// TwinCAT 3 PLC project Untitled1
// ProgramVersion: 3.1.4023.0
// libraries:
//   Tc2_Standard, * (Beckhoff Automation GmbH)
//   Tc2_System, * (Beckhoff Automation GmbH)
//   Tc3_Module, * (Beckhoff Automation GmbH)
// project tree:
//   / PlcTask.TcTTO
//   POUs/ FB_Flasher.TcPOU, MAIN.TcPOU, PRG_1.TcPOU
// real-time tasks:
//   TASK PlcTask: cycle T#10ms, priority 20, ADS port 350

CONFIGURATION Untitled1
    RESOURCE PLC ON TwinCAT3
        TASK PlcTask(INTERVAL := T#10ms, PRIORITY := 20);
        PROGRAM MAIN WITH PlcTask : MAIN;
    END_RESOURCE
END_CONFIGURATION

// ---- POUs/MAIN.TcPOU
PROGRAM MAIN
VAR

END_VAR



PRG_1();

END_PROGRAM

// ---- POUs/PRG_1.TcPOU
PROGRAM PRG_1
VAR
	
	nState: INT;	
	
	bSignalLamp: BOOL;
	
	bSelectorSw: BOOL;
	
	bMotorStart: BOOL;
	bMotorStop: BOOL;
	
	bMotor: BOOL;

	bDelta: BOOL;
	bStar: BOOL;

	bUp: BOOL;
	bDown: BOOL;
	bRight: BOOL;
	bLeft: BOOL;

	bMotorUp: BOOL;
	bMotorDown: BOOL;
	bMotorR: BOOL;
	bMotorL: BOOL;

	bUpSW: BOOL;
	bDownLW: BOOL;
	bRightSW: BOOL;
	bLeftSW: BOOL;
	
	bLedUp: BOOL;
	bLedDown: BOOL;
	bLedR: BOOL;
	bLedL: BOOL;
	
	FlasherRight: FB_Flasher;
	FlasherLeft: FB_Flasher;
	FlasherUp: FB_Flasher;
	FlasherDown: FB_Flasher;
	FB_FlasherCurrency: FB_Flasher;
	FB_FlasherTemp: FB_Flasher;
	
	T1: TON;
	T2: TON;
	
	nValue: INT;
	bFan1: BOOL;
	bFan2: BOOL;
	bTempLamp: BOOL;
	
	
	bEmergecyStop: BOOL;
	bCurrencyLamp: BOOL;
END_VAR



ACT_1();
ACT_3();

IF T2.Q THEN
	
	ACT_2();
			
END_IF



IF bEmergecyStop THEN
	//Her şeyi sıfırla
END_IF

ACTION ACT_1:

T1(IN:=bStar , PT:=T#2M , Q=> , ET=> );
T2(IN:=bMotor , PT:=T#5M , Q=> , ET=> );

CASE nState OF

	0:
	
		IF bSelectorSw THEN
			
			bSignalLamp	:=	TRUE;
			nState := 10;
			FB_FlasherCurrency(bStart:=FALSE);
			
		END_IF
	10:
	
		IF bMotorStart AND NOT bMotorStop THEN
			
			bStar	:=	TRUE;
			bDelta	:= FALSE;
			bMotor	:=	TRUE;
			
			nState := 20;
			
		END_IF
		
	20:	
	
		IF T1.Q THEN
			
			bStar	:=	FALSE;
			bDelta	:= 	TRUE;
			
		END_IF

END_CASE

IF NOT bMotorStart AND bMotorStop	THEN
	
	nState	:=	 0;
	bMotor	:=	FALSE;
	
END_IF

IF T1.Q AND NOT bUp 
AND NOT bDown 
AND NOT bRight
AND NOT bLeft THEN 

	FB_FlasherCurrency(bStart:=TRUE , bLed=>bCurrencyLamp );
	bMotor	:=	FALSE;
	nState	:=	0;
	
END_IF
END_ACTION

ACTION ACT_2:

//LimitSW ler NC olduğu kabul edilmiştir.

FlasherUp(bStart:=bMotorUp , bLed=>bLedUp );
FlasherDown(bStart:=bMotorDown , bLed=>bLedDown );

FlasherRight(bStart:=bMotorR , bLed=>bLedR );
FlasherLeft(bStart:=bMotorL , bLed=>bLedL );


IF bUp AND NOT bDown AND bUpSW THEN
	
	bMotorUp	:=	TRUE;
	bMotorDown	:=	FALSE;	
	
ELSIF bDown AND NOT bUp	AND bDownLW THEN
	
	bMotorUp	:=	FALSE;
	bMotorDown	:=	TRUE;
	
ELSIF	(bDown AND NOT bUp AND NOT bDownLW)
OR		(bUp AND NOT bDown AND NOT bUpSW) 	THEN
		
	bMotorUp	:=	FALSE;
	bMotorDown	:=	FALSE;	
	
END_IF



IF bRight AND NOT bLeft AND bRightSW THEN
	
	bMotorR	:=	TRUE;
	bMotorL	:=	FALSE;


ELSIF NOT bRight AND bLeft AND bLeftSW	THEN
	
	bMotorR	:=	FALSE;
	bMotorL	:=	TRUE;


ELSIF	(bRight	AND NOT bLeft AND NOT bRightSW)
OR 		(bLeft	AND NOT bRight AND NOT bLeftSW) THEN
		
	bMotorR	:=	FALSE;
	bMotorL	:=	FALSE;	
	
END_IF
END_ACTION

ACTION ACT_3:


FB_FlasherTemp(bStart:=bFan2, bLed=>bTempLamp );


IF nValue	>=	10 AND	nValue	<=	20 THEN		// Kademe_1
	
	bFan1	:=	TRUE;
	bFan2	:=	FALSE;
	
ELSIF	nValue > 20 THEN	//	Kademe_2
	
	bFan1	:=	TRUE;
	bFan2	:=	TRUE;
	
	bMotor	:=	FALSE;
	
	nState	:=	0;
	
END_IF
END_ACTION

END_PROGRAM

// ---- POUs/FB_Flasher.TcPOU
FUNCTION_BLOCK FB_Flasher
VAR_INPUT
		bStart: BOOL;
END_VAR
VAR_OUTPUT
	bLed: BOOL;
END_VAR
VAR
	nState: INT;
	TF1: TON;
	TF2: TON;
END_VAR



CASE nState	OF
	

	0:
		IF bStart THEN
			nState := 10;
		END_IF
		
	10:
	
		bLed	:=	TRUE;
	
		TF1(IN:=TRUE , PT:=T#500MS);
		
		IF TF1.Q THEN
			TF1(IN:=FALSE);
			nState := 20;
		END_IF
		
	20:
	
		bLed	:=	FALSE;
	
		TF2(IN:=TRUE , PT:=T#500MS);
		
		IF TF2.Q THEN
			TF2(IN:=FALSE);
			nState := 0;
		END_IF
		

END_CASE

END_FUNCTION_BLOCK
